Staubli VAL3: init.pgx

public program init()
begin
  nHandleCount=0
  bDebug=false
end
